FUNCTION_BLOCK FB_SelectorM3
VAR CONSTANT
    
END_VAR
VAR_INPUT
END_VAR
VAR_OUTPUT
END_VAR
VAR_IN_OUT
END_VAR
VAR
    
    stBaseIO : ST_M3DeviceBaseIO;

    stSelector	:	ST_SelectorM3;
    
    // Bronkhorst MFM
        stMFM	:	ST_BhElFlow;
    
    // Shakers
        {attribute 'pytmc' := '
            pv: Shaker1
         '}
        stShaker01	:	ST_Shaker;
        {attribute 'pytmc' := '
            pv: Shaker2
         '}
        stShaker02	:	ST_Shaker;
        {attribute 'pytmc' := '
            pv: Shaker3
         '}
        stShaker03	:	ST_Shaker;
        {attribute 'pytmc' := '
            pv: Shaker4
         '}
        stShaker04	:	ST_Shaker;
    
    // Vici valves
        fbSelectorSync	:	FB_SelectorSync;
        
        afbViciDriver : ARRAY [1..4] OF FB_ViciDriver;
        
        fbViciSerial  :   FB_SerialCommWrapper;
        stViciSerial  :   ST_SerialComm;
    
    //Sensirion flow meters
    {attribute 'pytmc' := '
        pv: SampleFM
     '}
	stSampleFM : ST_SensirionFM;
    
    {attribute 'pytmc' := '
        pv: SheathFM
     '}
	stSheathFM : ST_SensirionFM;
    
    astSelFM	: ARRAY[1..2] OF	ST_SensirionFM; //Address 1 is low flow, address 2 is high flow, low flow is mapped to M2 flow
	fbSensirionDriver	:	ARRAY [1..2] OF	FB_SensirionDriver;
    
    fbSensSerial : FB_SerialCommWrapper;
    stSensSerial : ST_SerialComm;

	stStatus: STRING;
	udCount: UDINT;

	tofReset: TOF;

	iIdOld	:	INT;
	
	viciIndex: INT := 1;
	fmIndex: INT;
    
    
    stComIn_EP6002P1		AT %I*	:	EL6inData22B (*KL6inData22B*);
	stComOut_EP6002P1		AT %Q*	:	EL6outData22B (*KL6outData22B*);

    
END_VAR

//Flowmeters
//////////////////////////////////////
Sensirion();

//Valve control
///////////////////////////////////
	fbSelectorSync(iq_stSelector:=stSelector);
	stSelector.stViciVlvCtrl[1].iReqPos := LIMIT(1, stSelector.iVici1ReqPos, 12);
	stSelector.stViciVlvCtrl[2].iReqPos := LIMIT(1, stSelector.iVici2ReqPos, 12);
	ViciDrivers();

	//for epics readback to be consistent
	IF stSelector.xResSyncd THEN stSelector.iSyncResPos := stSelector.stViciVlvStatus[1].iCurrPos; END_IF

(* Shakers *)
stShaker01.q_xPwrDO := stShaker01.i_xEpics;
stShaker02.q_xPwrDO := stShaker02.i_xEpics;
stShaker03.q_xPwrDO := stShaker03.i_xEpics;
stShaker04.q_xPwrDO := stShaker04.i_xEpics;

ACTION Sensirion:
(* Sensirion Flowmeter driver encapsulation*)

(* M3 selector has two flow meters. Sample and sheath. Sample is "low flow."*)

	
fbSensirionDriver[fmIndex](
	i_xExecute:= TRUE,
	i_tTimeOut:= t#1s,
	iq_stSerialRXBuffer:= stSensSerial.RxBuffer,
	iq_stSerialTXBuffer:= stSensSerial.TxBuffer,
	q_stStatus=>astSelFM[fmIndex].stat,
	i_stControl:=astSelFM[fmIndex].ctrl);

IF fbSensirionDriver[fmIndex].q_xDone OR
	fbSensirionDriver[fmIndex].q_xError OR
	fbSensirionDriver[fmIndex].q_xTimeout THEN

	
	IF fmIndex = 1 THEN 
		//Legacy flow
		//low flow maps to legacy readbacks
		stSampleFM.rFlow := astSelFM[fmIndex].stat.rFlow;
		stSampleFM.xFMOoR := astSelFM[fmIndex].stat.xOoR;
		stSampleFM.xFlowValid := astSelFM[fmIndex].stat.xFlowValid;
		stSampleFM.iFMState := astSelFM[fmIndex].stat.iState;
		stSampleFM.xFMModeRb := astSelFM[fmIndex].stat.xFMMode;
		//M3 flows
		stSelector.rLowFlow := astSelFM[fmIndex].stat.rFlow;
	ELSIF fmIndex = 2 THEN
		stSelector.rHighFlow := astSelFM[fmIndex].stat.rFlow;
	END_IF

	(* reset function for next time *)
	fbSensirionDriver[fmIndex].Reset();

	fmIndex := fmIndex + 1;
	IF fmIndex > 2 THEN fmIndex := 1;	END_IF
END_IF
END_ACTION

ACTION SerialComm:
fbSensSerial(stSerialComm := stSensSerial);
    
fbViciSerial(stSerialComm := stViciSerial);
END_ACTION

ACTION ViciDrivers:
afbViciDriver[viciIndex](
	i_xExecute:= TRUE,
	i_tTimeOut:= t#10s,
	i_stControl:= stSelector.stViciVlvCtrl[viciIndex],
	iq_stSerialRXBuffer:= stViciSerial.RxBuffer,
	iq_stSerialTXBuffer:= stViciSerial.TxBuffer,
	q_stStatus=>stSelector.stViciVlvStatus[viciIndex]);

IF 	afbViciDriver[viciIndex].q_xDone OR
	afbViciDriver[viciIndex].q_xError OR
	afbViciDriver[viciIndex].q_xTimeout THEN
	(* reset function for next time *)
	afbViciDriver[viciIndex](i_xExecute:=FALSE, 
        iq_stSerialRXBuffer:= stViciSerial.RxBuffer, 
        iq_stSerialTXBuffer:= stViciSerial.TxBuffer);
	
	viciIndex := viciIndex + 1;
	IF viciIndex > 2 THEN viciIndex := 1; END_IF
	
END_IF
END_ACTION

END_FUNCTION_BLOCK

(* stored: Version 1.1.0.1, ProductVersion 3.1.4022.18
   POU FB_SelectorM3: Id {a6869ee8-a1a6-4578-87e8-3c9673bf57ea}, SpecialFunc None
   Action Sensirion: Id {9f746844-7a59-4525-bff1-09e3ede82e12}
   Action SerialComm: Id {8e089361-fe69-4121-a86d-063809c21db5}
   Action ViciDrivers: Id {05c523af-4ae3-411a-b3b8-eed2754bd956} *)
